FUNCTION_BLOCK FB_ControllerType_1 EXTENDS FB_AbstructFuture
VAR_INPUT
END_VAR
VAR_OUTPUT
END_VAR
VAR
	_own_parameter: TIME;
	_set_time: TIME;
	process_timer: TON;
	blink_timer: TON;
	_result :UDINT;
	_own_output: REFERENCE TO BOOL;
END_VAR

METHOD abort : BOOL
IF process_timer.IN THEN
	_set_time := process_timer.PT - process_timer.ET;
END_IF
process_timer(IN := FALSE);
_own_output := FALSE;
abort := TRUE;
END_METHOD

METHOD execute : BOOL
VAR_INPUT
END_VAR
blink_timer(IN := NOT blink_timer.Q, PT := T#0.5S);
IF _own_output AND blink_timer.Q THEN
	_own_output := FALSE;
ELSIF blink_timer.Q THEN
	_own_output := TRUE;
END_IF
process_timer(IN := TRUE,PT := _set_time);
execute := process_timer.Q;
END_METHOD

METHOD init : BOOL
VAR_INPUT
END_VAR
_own_output := FALSE;
_set_time := _own_parameter;
process_timer(IN := FALSE);
blink_timer(IN := FALSE);
init := TRUE;
END_METHOD

PROPERTY nErrorID : UDINT
GET
END_GET
END_PROPERTY

PROPERTY own_output : REFERENCE TO BOOL
SET
_own_output REF= own_output;
END_SET
END_PROPERTY

PROPERTY own_parameter : TIME
GET
own_parameter := _own_parameter;
END_GET
SET
_own_parameter := own_parameter;
END_SET
END_PROPERTY

METHOD quit : BOOL
THIS^.init();
quit := TRUE;
END_METHOD

END_FUNCTION_BLOCK

(* stored: Version 1.1.0.1, ProductVersion 3.1.4024.12
   POU FB_ControllerType_1: Id {1076d71a-3a65-40e8-9c4e-a3e9e6fe7b78}, SpecialFunc None
   Method abort: Id {d02a02ce-eb9e-43cb-a107-d4fa0fc34c85}
   Method execute: Id {a437ddec-c1d7-448f-a879-d2b8cfc9472f}
   Method init: Id {67f09d3d-5c6c-4b82-bc02-bd0d47e41f54}
   Property nErrorID: Id {d940a05b-457a-4571-af02-9c908c0ddd5a}
   Get Get: Id {f38a3ee9-4b95-4da3-b87d-09c08cdf31f1}
   Property own_output: Id {2295a85b-9376-4fc8-b085-e01f4425b124}
   Set Set: Id {e86570c8-396d-4fc0-9e05-2ad72049042f}
   Property own_parameter: Id {da3dcd0a-6ea7-4769-9b14-2d35ed1ea4ae}
   Get Get: Id {91ea83f3-ac89-44fe-88f4-aaf098638ab9}
   Set Set: Id {6598af7b-282d-427f-83dd-91a46e26192a}
   Method quit: Id {906e42c6-5cb2-4ee4-be39-84be0bedded2} *)
